PROGRAM MAIN
VAR
	XPlanarTable  : FB_Component_XPlanar;
	Mover		  : FB_XPlanarMover;
	i			  : UDINT;
	EnableMovers  : BOOL;
	DisableMovers : BOOL;
	MoveCmd1	  : BOOL;
	MoveCmd2	  : BOOL;
	CommandResult : I_PlanarTaskResult;
END_VAR

//Set the intefaces for background functions **This must be done first!**
ip.Movers[1] := Mover;

//Keep the XPlanar System up to date
XplanarTable.CyclicLogic();

//Enable movers
IF EnableMovers THEN
	IF Mover.Enable().Done THEN
		EnableMovers := FALSE; 
	END_IF
END_IF

//DisableMovers
IF DisableMovers THEN
	IF Mover.Disable().Done THEN
		DisableMovers := FALSE;
	END_IF
END_IF

//Move 1
IF MoveCmd1 THEN
	IF Mover.MoveCommand.FreeMove(120, 360).Done THEN
		MoveCmd1 := FALSE;
	END_IF
END_IF

//Move 2
IF MoveCmd2 THEN
	IF Mover.MoveCommand.FreeMove(120, 120).Done THEN
		MoveCmd2 := FALSE;
	END_IF	
END_IF

END_PROGRAM

(* stored: Version 1.1.0.1, ProductVersion 3.1.4024.13
   POU MAIN: Id {ac785b93-3788-4896-9f9d-1a7a58c51c67}, SpecialFunc None *)
